// TIA Portal V21 export
VAR_GLOBAL   // PLC tag table "UnitaDiMisura_Grandezze"
END_VAR
VAR_GLOBAL CONSTANT   // user constants
   Um_Grandezza_Lunghezza : Int := 1;
   Um_Grandezza_Tempo : Int := 2;
   Um_Grandezza_Temperatura : Int := 3;
   Um_Grandezza_Percentuale : Int := 4;
   Um_Grandezza_Portata : Int := 5;
   Um_Grandezza_Concentrazione : Int := 7;
   Um_Grandezza_Pressione : Int := 6;
END_VAR
